% RSLogix 500 project P3_ABIOLA_A_V2_BAK006.RSS, saved by version 8.30.00.16 %
PROJECT "UNTITLED"    % processor: Bul.1763 MicroLogix 1100 Series B %

PROGRAM FILES
  LAD 2   2 rungs
  LAD 3 "PSEUDO IO"  4 rungs  % Contains all the assigned memery address used  %

DATA FILES
  O0 OUTPUT  4 elements
  I1 INPUT  6 elements
  S2 STATUS  66 elements
  B3 BINARY  1 elements
  T4 TIMER  1 elements
  C5 COUNTER  1 elements
  R6 CONTROL  1 elements
  N7 INTEGER  3 elements
  F8 FLOAT  1 elements
  ST9 STRFRBCSCN  1 elements  % Writes string from bar code scanner to PLC %

LADDER 2
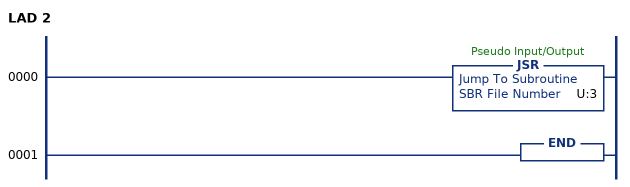
% Rung: 0 %
SOR JSR U:3 EOR
%   U:3  "Pseudo Input/Output" %
% Rung: 1 %
SOR END EOR

LADDER 3 "PSEUDO IO"    % Contains all the assigned memery address used  %
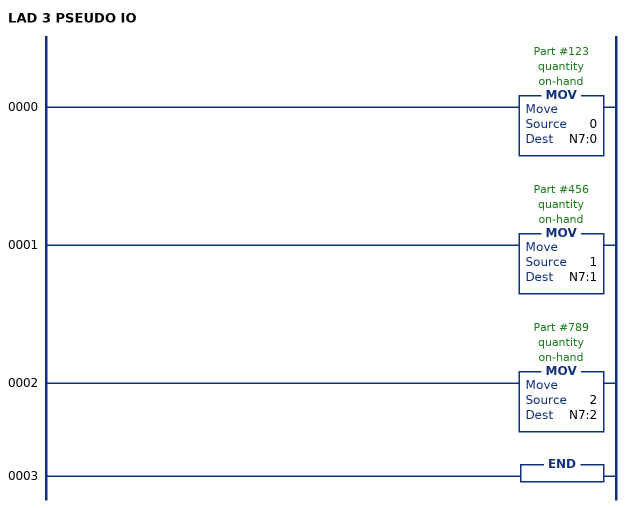
% Rung: 0 %
SOR MOV 0 N7:0 EOR
%   N7:0  "Part #123 quantity on-hand" %
% Rung: 1 %
SOR MOV 1 N7:1 EOR
%   N7:1  "Part #456 quantity on-hand" %
% Rung: 2 %
SOR MOV 2 N7:2 EOR
%   N7:2  "Part #789 quantity on-hand" %
% Rung: 3 %
SOR END EOR
